{attribute 'GeneratedUsingTerminal: EK1122-0000-0018'}
{attribute addProperty BoxType "EK1122-0000-0018"}
{attribute addProperty Id "Beckhoff_EJ4xxxsub_EK1100EK1100_AB5A94672"}
{attribute addProperty CRC "253848064"}
{attribute addProperty Size "2"}
TYPE Beckhoff_EJ4xxxEK1122_0F216A00 EXTENDS EK1122_AB5A9467 :
STRUCT
	{attribute addProperty Name "Beckhoff_EJ4xxxsub_EK1100"}
	{attribute addProperty PreviousPort "Beckhoff EJ4xxxEK1122 : D"}
	Beckhoff_EJ4xxxsub_EK1100 : EK1100_AB5A9467;
END_STRUCT
END_TYPE

(* stored: Version 1.2.0.0, ProductVersion 3.1.4024.9
   DUT Beckhoff_EJ4xxxEK1122_0F216A00: Id {a3bacbf7-5db1-4d5e-8577-ae48fbabf501} *)
